# EPICS autosave request: apps/xpsMotorApp/Db/motorsTaggerHall.req
$(PREF)T1-7-BOT:m6:scan1.P1PA
$(PREF)T1-7-BOT:m6:scan1.P1SM
$(PREF)T1-7-BOT:m6:scan1.P1SP
$(PREF)T1-7-BOT:m6:scan1.P1EP
$(PREF)T1-7-BOT:m6:scan1.NPTS
$(PREF)T1-7-BOT:m6:saveData_scanNumber
$(PREF)T1-7-BOT:m6:saveData_fileSystem
$(PREF)T1-7-BOT:m6:saveData_subDir
$(PREF)T1-7-BOT:m6:saveData_baseName
$(PREF)T1-7-BOT:m6:scan1.PDLY
$(PREF)T1-7-BOT:m6:scan1.DDLY
